FUNCTION_BLOCK "FB_test"
{ S7_Optimized_Access := 'TRUE' }


VAR_INPUT
END_VAR

VAR

END_VAR

BEGIN


END_FUNCTION_BLOCK